PROGRAM PRG_PC5K4
VAR
    {attribute 'pytmc' :='pv: PC5K4:FWM'}
    {attribute 'TcLinkTo' := '.fbFlowMeter.iRaw := TIIB[EP3174-FWM-E2]^AI Standard Channel 1^Value'}
    fbFlowMeter: FB_FDQ_FlowMeter;
END_VAR

fbFlowMeter();

END_PROGRAM

(* stored: Version 1.1.0.1, ProductVersion 3.1.4024.12
   POU PRG_PC5K4: Id {239e0261-00ca-4d33-8394-23cf4a49ddc7}, SpecialFunc None *)
